FUNCTION_BLOCK Command_to_Action
VAR_INPUT
	inputString : STRING;
END_VAR
VAR_OUTPUT
	recognitionValue : REAL;
	Busy : BOOL;
END_VAR
VAR
	putString : STRING;
	recognitionString : STRING := 'Steer(';
	stringLength : int;
END_VAR

inputString := GetSpeedSteer.steerString;

Busy := FALSE;
IF GetSpeedSteer.bExecuteSteer THEN
	Busy := TRUE;
END_IF

IF FIND(STR1:= inputString  , STR2:= recognitionString ) = 1 THEN
	putString := DELETE(STR:=inputString , LEN:= 6 , POS:=1 );
	stringLength := LEN(putstring);
	putString := DELETE(STR:=putString , LEN:= 1 , POS:= stringLength);
	recognitionValue := STRING_TO_INT(putString);
END_IF

END_FUNCTION_BLOCK

(* stored: Version 1.1.0.1, ProductVersion 3.1.4024.3
   POU Command_to_Action: Id {ae358f74-febb-409c-b913-83a08ed40d1a}, SpecialFunc None *)
